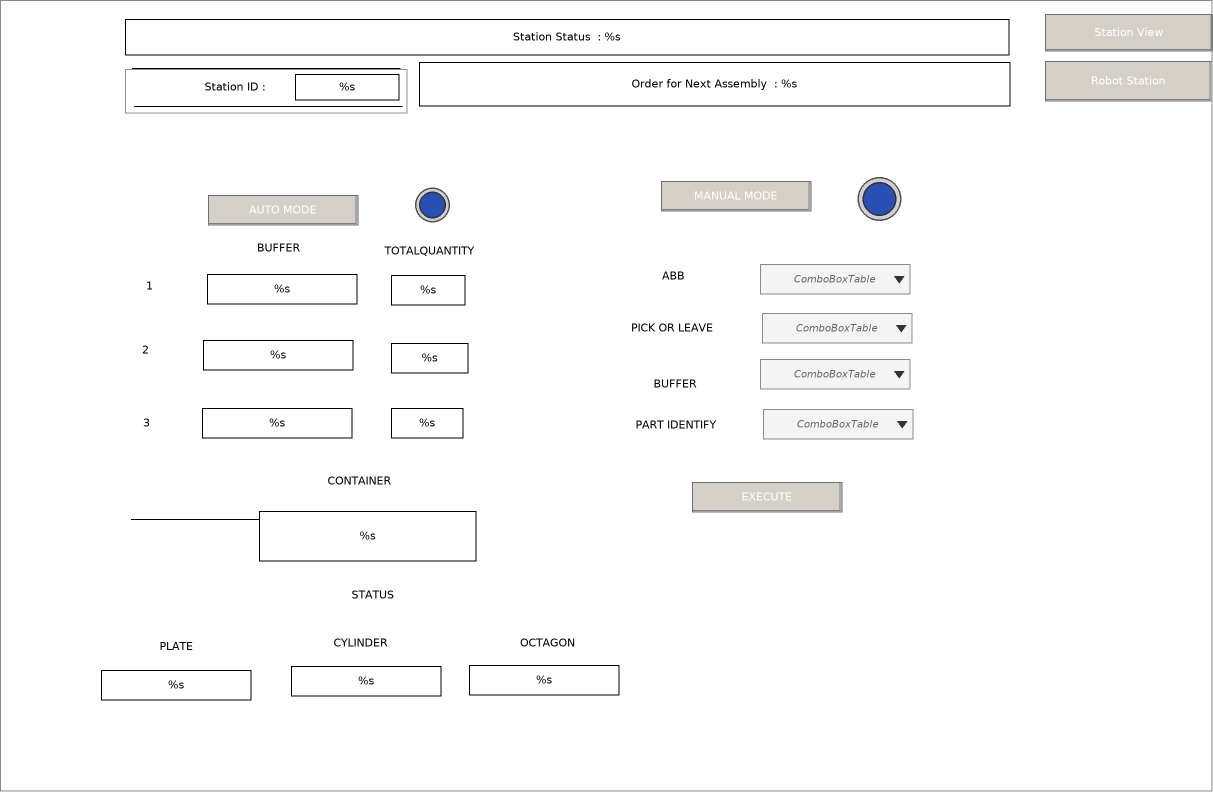
VISUALIZATION Visualization  // 1213x792
    Rectangle (125,19 884x36), "Station Status : %s", text variable: Visualaisation_Control.mxStationStatus
    GroupBox (125,61 282x52)
        Line (6,458) (274,458)
        Line (7,7) (275,7)
        Label (35,11 150x30), "Station ID :"
        Rectangle (170,13 104x26), "%s", text variable: GVL.mwStationID
        Line (9,45) (277,45)
    Button (1045,61 167x40), "Robot Station"
        OnMouseClick: change screen: RobotStation
    Rectangle (419,62 591x44), "Order for Next Assembly : %s", text variable: GVL.qsOrderFornextAssembly
    Button (1045,14 168x37), "Station View"
        OnMouseClick: change screen: Station
    Lamp1 (408,185 49x40), variable: ModeControl.AutoMode, style: Lamp-Lamp1-Blue
    Lamp1 (854,173 51x52), variable: ModeControl.ManualMode, style: Lamp-Lamp1-Blue
    Label (232,233 93x30), "BUFFER"
    Textfield (207,274 150x30), "%s", text variable: GVL.BufferProducts.Storage1.Component
    Label (367,236 125x30), "TOTALQUANTITY"
    Textfield (203,340 150x30), "%s", text variable: GVL.BufferProducts.Storage2.Component
    Textfield (202,408 150x30), "%s", text variable: GVL.BufferProducts.Storage3.Component
    Textfield (391,275 74x30), "%s", text variable: GVL.BufferProducts.Storage1.Quatity
    Textfield (391,343 77x30), "%s", text variable: GVL.BufferProducts.Storage2.Quatity
    Textfield (391,408 72x30), "%s", text variable: GVL.BufferProducts.Storage3.Quatity
    Textfield (259,511 217x50), "%s", text variable: LoadFromAGV.ContainerColor
    Label (133,271 33x30), "1"
    Label (129,335 33x30), "2"
    Label (130,408 33x30), "3"
    Label (296,466 127x30), "CONTAINER"
    Label (118,625 117x43), "PLATE"
    Label (314,628 93x30), "CYLINDER"
    Label (501,628 93x30), "OCTAGON"
    Label (267,575 212x40), "STATUS"
    Label (600,261 150x30), "ABB"
    Label (597,313 150x30), "PICK OR LEAVE"
    Label (600,369 150x30), "BUFFER"
    Label (601,410 150x30), "PART IDENTIFY"
    Label (650,762 150x30)
    Textfield (101,670 150x30), "%s", text variable: AssembleParts.AssembledParts[1]
    Textfield (291,666 150x30), "%s", text variable: AssembleParts.AssembledParts[2]
    Textfield (469,665 150x30), "%s", text variable: AssembleParts.AssembledParts[3]
    Button (692,482 150x30), "EXECUTE"
        tap ManualMode.Execute
    Button (661,181 150x30), "MANUAL MODE"
        tap ModeControl.ManualModeButtonClick
    Button (208,195 150x30), "AUTO MODE"
        tap ModeControl.AutoModeButtonClick
    ComboBoxTable (760,264 150x30), variable: ManualMode.ABBFunction, data array: GVL.sABBFunction
        p3854506369: GVL.sABBFunction[INDEX]
    ComboBoxTable (762,313 150x30), variable: ManualMode.PickLeave, data array: GVL.sPickOrLeave
        p3854506369: GVL.sPickOrLeave[INDEX]
    ComboBoxTable (760,359 150x30), variable: ManualMode.BufferID, data array: GVL.sBufferIDlist
        p3854506369: GVL.sBufferIDlist[INDEX]
    ComboBoxTable (763,409 150x30), variable: ManualMode.Part, data array: GVL.sPart
        p3854506369: GVL.sPart[INDEX]
END_VISUALIZATION

(* stored: Version 1.1.0.1, ProductVersion 3.1.4024.12
   Visu Visualization: Id {08c1f753-3e44-4c26-b458-35ef78727ab8} *)
